// TwinCAT 3 PLC project StudentStation
// ProgramVersion: 3.1.4022.4
// libraries:
//   Tc2_Standard, * (Beckhoff Automation GmbH)
//   Tc2_System, * (Beckhoff Automation GmbH)
//   Tc3_Module, * (Beckhoff Automation GmbH)
//   VisuDialogs, * (System)
//   VisuSymbols,3.5.10.0,System
// project tree:
//   ABBControl/ ABBAssemble.TcPOU (not stored), ABBGotoAGVPos.TcPOU (not stored), ABBGotoBuffer.TcPOU (not stored), ABBGotoHome.TcPOU (not stored), ABBGotoScanner.TcPOU (not stored), ABBGotoTable.TcPOU (not stored), ABBPickLeaveBuffer.TcPOU (not stored), ABBPickLeaveContainerAGV.TcPOU (not stored), ABBPickLeaveContaineronTable.TcPOU (not stored), ABBPickLeaveScanner.TcPOU (not stored), ABBScanContainer.TcPOU (not stored), ABBScannerStation.TcPOU (not stored)
//   Automation Library/ AGVControlSystem.TcPOU (not stored), AutomationLibrary.TcPOU (not stored), BookingSystem.TcPOU (not stored), CommData.TcGVL (not stored), OrderHandling.TcPOU (not stored), PhysicalSystemTest.TcPOU (not stored), RobotControlSystem.TcPOU (not stored), RobotPosTracker.TcPOU (not stored), SensorReader.TcPOU (not stored), Visualaisation_Control.TcPOU (not stored)
//   DUTs/ ABBPositions.TcDUT (not stored), ABBXYPOS.TcDUT (not stored), OrderPLC.TcDUT (not stored), PLCRobotOrder.TcDUT (not stored), Station.TcDUT (not stored), Storage.TcDUT (not stored)
//   / GlobalTextList.TcGTLO, PlcTask.TcTTO (not stored), Visualization Manager.TcVMO (not stored)
//   GVLs/ GVL.TcGVL
//   POUs/ ModeControl.TcPOU, ManualMode.TcPOU, AssembleParts.TcPOU, LoadFromAGV.TcPOU, ScanBuffer.TcPOU, Robot.TcPOU, AutoMode.TcPOU, MAIN.TcPOU, IdentifyPart.TcPOU
//   VISUs/ RobotStation.TcVIS (not stored), Station.TcVIS, Visualization.TcVIS
// real-time tasks:
//   TASK PlcTask: cycle T#10ms, priority 20, ADS port 350

// ---- GVLs/GVL.TcGVL
{attribute 'qualified_only'}
VAR_GLOBAL
	// Order for the next assembly part. The part name should be sent as per the part list and case sensitive. 
	{attribute 'OPC.UA.DA' := '1'}
	qsOrderFornextAssembly AT %Q*: STRING := '0';
	// Parts in your Station buffer. Each buffer have 3 storage locations. The part name and quantity should be mentioned.
	{attribute 'OPC.UA.DA' := '1'}
	BufferProducts AT %Q*: Station;
	// Signal to AGV, a pallet is placed from Station to the AGV. 
	{attribute 'OPC.UA.DA' := '1'}
	qxPalletPlacedinAGV AT %Q*: BOOL;
	// Signal From AGV, that it have docked in your station
	{attribute 'OPC.UA.DA' := '1'}
	ixAGVatStation AT %I*: BOOL;
	// Signal Denoting An AGV have arrived in the Station
	{attribute 'OPC.UA.DA' := '1'}	
	qxPickedfromAGV AT %Q*:BOOL; //Part is picked up from the AGV
	{attribute 'OPC.UA.DA' := '1'}
	mwStationStatus AT %Q*: INT; //Pre-Conditioning Mode //100:Ready to Work § 200: Getting Booked § 300: Booked and Busy § 400 : Manual mode  § 500: Pause Mode § 1000 : Emergency Mode 
	{attribute 'OPC.UA.DA' := '1'}	
	// Emergency Stop is active
	ixEmergencyStop AT %Q*:BOOL;
	
	// Inductive sensor reading. from scaning station
	ixInductiveSensor1 AT %I*:BOOL;
	// Inductive sensor reading. from scaning station
	ixInductiveSensor2 AT %I*:BOOL;
	// Inductive sensor reading. from scaning station
	ixInductiveSensor3 AT %I*:BOOL;
	// Inductive sensor reading. from scaning station
	ixInductiveSensor4 AT %I*:BOOL;
	// Inductive sensor reading. from the sensor in robot Tool
	ixInductiveSensorinTool AT %I*:BOOL;
	// Station ID of the station you are working with.
	{attribute 'OPC.UA.DA' := '1'}
	mwStationID AT %Q*: INT;
	
	sABBFunction : ARRAY [1..12] OF STRING := ['ABBAssemble','ABBGotoAGVPos','ABBGotoBuffer','ABBGotoHome','ABBGotoScanner','ABBGotoTable','ABBPickLeaveBuffer','ABBPickLeaveContainerAGV','ABBPickLeaveContainerOnTable','ABBPickLeaveScanner','ABBScanContainer', 'ABBScannerStation'];
	sBufferIDlist : ARRAY [1..3] OF STRING := ['Storage Position 1','Storage Position 2','Storage Position 3'];
	sPart : ARRAY [1..3] OF STRING := ['Plate','Cylinder','Octagon'];
	sPickOrLeave : ARRAY [1..2] OF STRING := ['Pick','Leave'];
	sABBFunctionList : ARRAY [1..12] OF STRING := ['ABBAssemble','ABBGotoAGVPos','ABBGotoBuffer','ABBGotoHome','ABBGotoScanner','ABBGotoTable','ABBPickLeaveBuffer','ABBPickLeaveContainerAGV','ABBPickLeaveContainerOnTable','ABBPickLeaveScanner','ABBScanContainer', 'ABBScannerStation'];
END_VAR

// ---- POUs/Robot.TcPOU
PROGRAM Robot
VAR
	// Goto Home
	ABBGotoHome_Control: ABBGotoHome;
	GotoHome: BOOL;
	GotoHomeDone: BOOL;
	
	// Go to AGV
	ABBGotoAGVPosByScanner_Control: ABBGotoAGVPos;
	GotoAGVByScanner: BOOL;
	GotoAGVByScannerDone: BOOL;
	
	// Go to AGV
	ABBGotoAGVPosByAssembly_Control: ABBGotoAGVPos;
	GotoAGVByAssembly: BOOL;
	GotoAGVByAssemblyDone: BOOL;
	
	// Go to Scanner
	ABBGotoScannerFromAGV_Control: ABBGotoScanner;
	ABBGotoScannerFromBuffer_Control: ABBGotoScanner;
	GotoScannerFromBuffer: BOOL;
	GotoScannerFromAGV: BOOL;
	GotoScannerFromBufferDone: BOOL;
	GotoScannerFromAGVDone: BOOL;
	
	// Go to Table
	ABBGotoTableByAGV_Control: ABBGotoTable;
	GotoTableByAGV: BOOL;
	GotoTableByAGVDone: BOOL;
	
	ABBGotoTableByScanner_Control: ABBGotoTable;
	GotoTableByScanner: BOOL;
	GotoTableDoneByScanner: BOOL;
	
	ABBGotoTableByAssembly_Control: ABBGotoTable;
	GotoTableByAssembly: BOOL;
	GotoTableDoneByAssembly: BOOL;
	
	// Go to Buffer
	ABBGotoBuffer_Control: ABBGotoBuffer;
	GotoBuffer: BOOL;
	GotoBufferDone: BOOL;
	
	// PickLeave Container AGV
	ABBPickLeaveContainerAGV_Control: ABBPickLeaveContainerAGV;
	PickAGV: BOOL;
	LeaveAGV: BOOL;
	PickLeaveAGVDone: BOOL;
	
	// PickLeave Scanner
	ABBPickLeaveScannerFromBuffer_Control: ABBPickLeaveScanner;
	ABBPickLeaveScannerFromAGV_Control: ABBPickLeaveScanner;
	PickScannerFromBuffer: BOOL;
	LeaveScannerFromBuffer: BOOL;
	PickLeaveScannerFromBufferDone: BOOL;
	PickScannerFromAGV: BOOL;
	LeaveScannerFromAGV: BOOL;
	PickLeaveScannerFromAGVDone: BOOL;
	
	
	// PickLeave Buffer
	ABBPickLeaveBuffer_Control: ABBPickLeaveBuffer;
	PickBuffer: BOOL;
	LeaveBuffer: BOOL;
	PickLeaveBufferDone: BOOL;
	
	// PickLeave Table
	ABBPickLeaveTable_Control: ABBPickLeaveContaineronTable;
	PickTable: BOOL;
	LeaveTable: BOOL;
	PickLeaveTableDone: BOOL;
	
	// Scan parts
	ABBScanContainer_Control: ABBScanContainer;
	ScanContainer: BOOL;
	ScanContainerPartAvailable: BOOL;
	ScanContainerDone: BOOL;
	
	// Assemble parts
	ABBAssemble_Control: ABBAssemble;
	Assemble: BOOL;
	AssembleBufferId: INT;
	AssemblePartId: INT;
	AssembleDone: BOOL;
	
	// Read sensor
	ABBScannerStationByBuffer_Control: ABBScannerStation;
	ABBScannerStationByAGV_Control: ABBScannerStation;
	ReadSensorByBuffer: BOOL;
	ReadSensorByAGV: BOOL;
	ReadSensorByBufferDone: BOOL;
	ReadSensorByAGVDone: BOOL;
	
	
	// Read sensor
	IdentifyPartFB: IdentifyPart;
	IdentifyPart_Control: IdentifyPart;
	ScanPartId: INT;
END_VAR

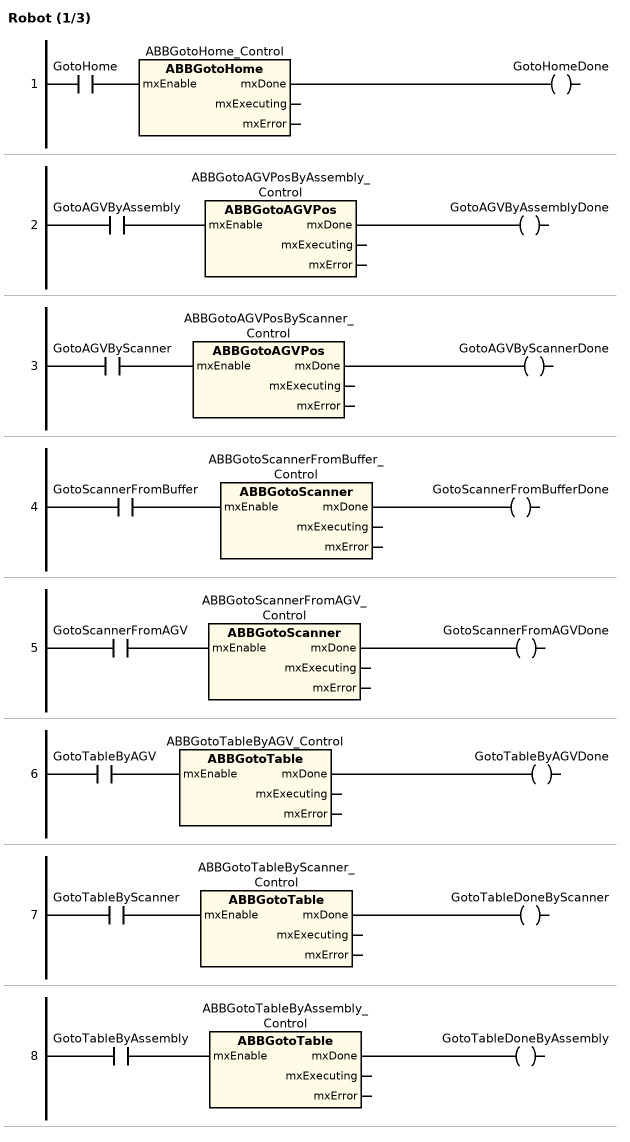
// NETWORK 1
ABBGotoHome_Control(mxEnable := GotoHome); // ABBGotoHome
GotoHomeDone := ABBGotoHome_Control.mxDone;

// NETWORK 2
ABBGotoAGVPosByAssembly_Control(mxEnable := GotoAGVByAssembly); // ABBGotoAGVPos
GotoAGVByAssemblyDone := ABBGotoAGVPosByAssembly_Control.mxDone;

// NETWORK 3
ABBGotoAGVPosByScanner_Control(mxEnable := GotoAGVByScanner); // ABBGotoAGVPos
GotoAGVByScannerDone := ABBGotoAGVPosByScanner_Control.mxDone;

// NETWORK 4
ABBGotoScannerFromBuffer_Control(mxEnable := GotoScannerFromBuffer); // ABBGotoScanner
GotoScannerFromBufferDone := ABBGotoScannerFromBuffer_Control.mxDone;

// NETWORK 5
ABBGotoScannerFromAGV_Control(mxEnable := GotoScannerFromAGV); // ABBGotoScanner
GotoScannerFromAGVDone := ABBGotoScannerFromAGV_Control.mxDone;

// NETWORK 6
ABBGotoTableByAGV_Control(mxEnable := GotoTableByAGV); // ABBGotoTable
GotoTableByAGVDone := ABBGotoTableByAGV_Control.mxDone;

// NETWORK 7
ABBGotoTableByScanner_Control(mxEnable := GotoTableByScanner); // ABBGotoTable
GotoTableDoneByScanner := ABBGotoTableByScanner_Control.mxDone;

// NETWORK 8
ABBGotoTableByAssembly_Control(mxEnable := GotoTableByAssembly); // ABBGotoTable
GotoTableDoneByAssembly := ABBGotoTableByAssembly_Control.mxDone;

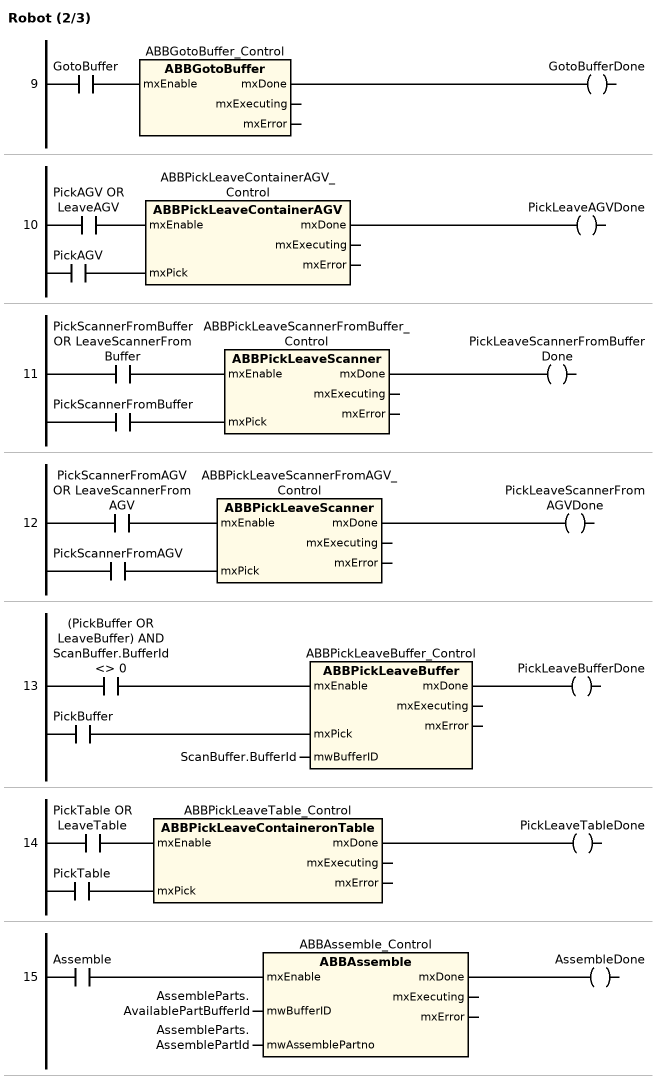
// NETWORK 9
ABBGotoBuffer_Control(mxEnable := GotoBuffer); // ABBGotoBuffer
GotoBufferDone := ABBGotoBuffer_Control.mxDone;

// NETWORK 10
ABBPickLeaveContainerAGV_Control(mxEnable := PickAGV OR LeaveAGV, mxPick := PickAGV); // ABBPickLeaveContainerAGV
PickLeaveAGVDone := ABBPickLeaveContainerAGV_Control.mxDone;

// NETWORK 11
ABBPickLeaveScannerFromBuffer_Control(mxEnable := PickScannerFromBuffer OR LeaveScannerFromBuffer, mxPick := PickScannerFromBuffer); // ABBPickLeaveScanner
PickLeaveScannerFromBufferDone := ABBPickLeaveScannerFromBuffer_Control.mxDone;

// NETWORK 12
ABBPickLeaveScannerFromAGV_Control(mxEnable := PickScannerFromAGV OR LeaveScannerFromAGV, mxPick := PickScannerFromAGV); // ABBPickLeaveScanner
PickLeaveScannerFromAGVDone := ABBPickLeaveScannerFromAGV_Control.mxDone;

// NETWORK 13
ABBPickLeaveBuffer_Control(
    mxEnable := (PickBuffer OR LeaveBuffer) AND ScanBuffer.BufferId <> 0,
    mxPick := PickBuffer,
    mwBufferID := ScanBuffer.BufferId); // ABBPickLeaveBuffer
PickLeaveBufferDone := ABBPickLeaveBuffer_Control.mxDone;

// NETWORK 14
ABBPickLeaveTable_Control(mxEnable := PickTable OR LeaveTable, mxPick := PickTable); // ABBPickLeaveContaineronTable
PickLeaveTableDone := ABBPickLeaveTable_Control.mxDone;

// NETWORK 15
ABBAssemble_Control(
    mxEnable := Assemble,
    mwBufferID := AssembleParts.AvailablePartBufferId,
    mwAssemblePartno := AssembleParts.AssemblePartId); // ABBAssemble
AssembleDone := ABBAssemble_Control.mxDone;

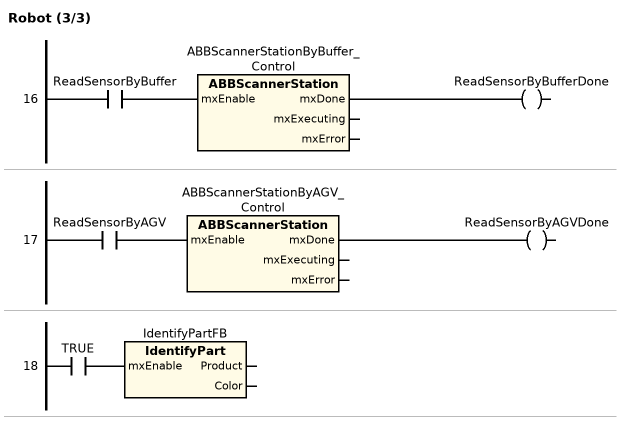
// NETWORK 16
ABBScannerStationByBuffer_Control(mxEnable := ReadSensorByBuffer); // ABBScannerStation
ReadSensorByBufferDone := ABBScannerStationByBuffer_Control.mxDone;

// NETWORK 17
ABBScannerStationByAGV_Control(mxEnable := ReadSensorByAGV); // ABBScannerStation
ReadSensorByAGVDone := ABBScannerStationByAGV_Control.mxDone;

// NETWORK 18
IdentifyPartFB(mxEnable := TRUE); // IdentifyPart

END_PROGRAM

// ---- POUs/IdentifyPart.TcPOU
FUNCTION_BLOCK IdentifyPart
VAR_INPUT
	mxEnable: BOOL;
END_VAR
VAR_OUTPUT
	Product:STRING;
	Color: STRING;
	Component: STRING;
END_VAR
VAR
	SensorReader:BYTE;
END_VAR

IF mxEnable THEN
	SensorReader.1:=gvl.ixInductiveSensor1;
	SensorReader.2:=gvl.ixInductiveSensor2;
	SensorReader.3:=gvl.ixInductiveSensor3;
	SensorReader.4:=gvl.ixInductiveSensor4;
END_IF

IF SensorReader = 0 OR SensorReader = 4 OR SensorReader = 2 OR SensorReader = 6 THEN
 	Product:='InvalidPart';
	Color := '';
	Component := 'invalidpart';
END_IF

IF SensorReader=16 THEN
	Product:='CONTAINER';
	Color := 'BLUE';
	Component := 'BLUECONTAINER';
END_IF

IF SensorReader=8 THEN
	Product:='CONTAINER';
	Color := 'YELLOW';
	Component := 'YELLOWCONTAINER';
END_IF

IF SensorReader=24 THEN
	Product:='CONTAINER';
	Color := 'RED';
	Component := 'REDCONTAINER';
END_IF

IF SensorReader=20 THEN
	Product:='CYLINDER';
	Color := 'BLUE';
	Component := 'BLUECYLINDER';
END_IF

IF SensorReader=12 THEN
	Product:='OCTAGON';
	Color := 'BLUE';
	Component := 'BLUEOCTAGON';
END_IF

IF SensorReader=28 THEN
	Product:='PLATE';
	Color := 'BLUE';
	Component := 'BLUEPLATE';
END_IF

IF SensorReader=18 THEN
	Product:='CYLINDER';
	Color := 'YELLOW';
	Component := 'YELLOWCYLINDER';
END_IF

IF SensorReader=10 THEN
	Product:='OCTAGON';
	Color := 'YELLOW';
	Component := 'YELLOWOCTAGON';
END_IF

IF SensorReader=26 THEN
	Product:='PLATE';
	Color := 'YELLOW';
	Component := 'YELLOWPLATE';
END_IF

IF SensorReader=22 THEN
	Product:='CYLINDER';
	Color := 'RED';
	Component := 'REDCYLINDER';
END_IF

IF SensorReader=14 THEN
	Product:='OCTAGON';
	Color := 'RED';
	Component := 'REDOCTAGON';
END_IF

IF SensorReader=30 THEN
	Product:='PLATE';
	Color := 'RED';
	Component := 'REDPLATE';
END_IF

END_FUNCTION_BLOCK

// ---- POUs/ScanBuffer.TcPOU
PROGRAM ScanBuffer
VAR
	// Default
	Done: BOOL;
	
	// Goto Buffer id
	BufferId: INT;
	BufferIdReady: BOOL;
	
	// Invalid Buffer part
	InvalidPart: BOOL;
	Quatity: INT;
END_VAR

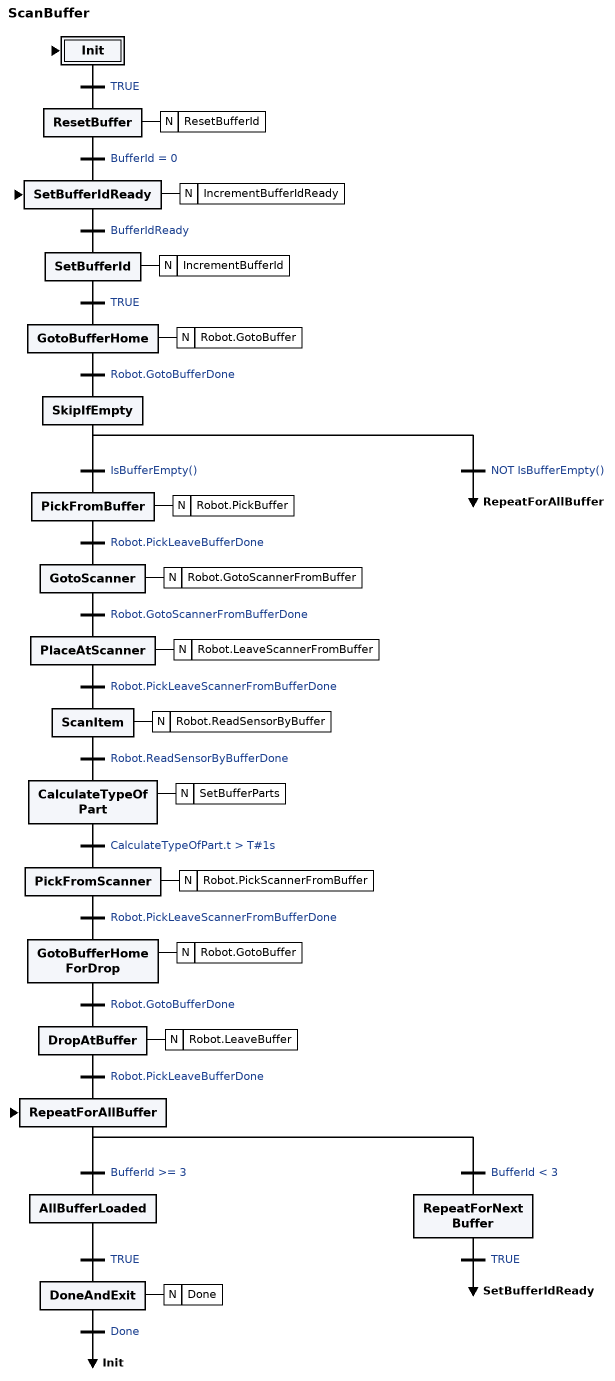
INITIAL_STEP Init:
END_STEP
TRANSITION FROM Init TO ResetBuffer
    := TRUE;
END_TRANSITION
STEP ResetBuffer:
    ResetBufferId(N);
END_STEP
TRANSITION FROM ResetBuffer TO SetBufferIdReady
    := BufferId = 0;
END_TRANSITION
STEP SetBufferIdReady:
    IncrementBufferIdReady(N);
END_STEP
TRANSITION FROM SetBufferIdReady TO SetBufferId
    := BufferIdReady;
END_TRANSITION
STEP SetBufferId:
    IncrementBufferId(N);
END_STEP
TRANSITION FROM SetBufferId TO GotoBufferHome
    := TRUE;
END_TRANSITION
STEP GotoBufferHome:
    Robot.GotoBuffer(N);
END_STEP
TRANSITION FROM GotoBufferHome TO SkipIfEmpty
    := Robot.GotoBufferDone;
END_TRANSITION
STEP SkipIfEmpty:
END_STEP
TRANSITION FROM SkipIfEmpty TO PickFromBuffer
    := IsBufferEmpty();
END_TRANSITION
TRANSITION FROM SkipIfEmpty TO RepeatForAllBuffer
    := NOT IsBufferEmpty();
END_TRANSITION
STEP PickFromBuffer:
    Robot.PickBuffer(N);
END_STEP
TRANSITION FROM PickFromBuffer TO GotoScanner
    := Robot.PickLeaveBufferDone;
END_TRANSITION
STEP GotoScanner:
    Robot.GotoScannerFromBuffer(N);
END_STEP
TRANSITION FROM GotoScanner TO PlaceAtScanner
    := Robot.GotoScannerFromBufferDone;
END_TRANSITION
STEP PlaceAtScanner:
    Robot.LeaveScannerFromBuffer(N);
END_STEP
TRANSITION FROM PlaceAtScanner TO ScanItem
    := Robot.PickLeaveScannerFromBufferDone;
END_TRANSITION
STEP ScanItem:
    Robot.ReadSensorByBuffer(N);
END_STEP
TRANSITION FROM ScanItem TO CalculateTypeOfPart
    := Robot.ReadSensorByBufferDone;
END_TRANSITION
STEP CalculateTypeOfPart:
    SetBufferParts(N);
END_STEP
TRANSITION FROM CalculateTypeOfPart TO PickFromScanner
    := CalculateTypeOfPart.t > T#1s;
END_TRANSITION
STEP PickFromScanner:
    Robot.PickScannerFromBuffer(N);
END_STEP
TRANSITION FROM PickFromScanner TO GotoBufferHomeForDrop
    := Robot.PickLeaveScannerFromBufferDone;
END_TRANSITION
STEP GotoBufferHomeForDrop:
    Robot.GotoBuffer(N);
END_STEP
TRANSITION FROM GotoBufferHomeForDrop TO DropAtBuffer
    := Robot.GotoBufferDone;
END_TRANSITION
STEP DropAtBuffer:
    Robot.LeaveBuffer(N);
END_STEP
TRANSITION FROM DropAtBuffer TO RepeatForAllBuffer
    := Robot.PickLeaveBufferDone;
END_TRANSITION
STEP RepeatForAllBuffer:
END_STEP
TRANSITION FROM RepeatForAllBuffer TO AllBufferLoaded
    := BufferId >= 3;
END_TRANSITION
STEP AllBufferLoaded:
END_STEP
TRANSITION FROM AllBufferLoaded TO DoneAndExit
    := TRUE;
END_TRANSITION
TRANSITION FROM RepeatForAllBuffer TO RepeatForNextBuffer
    := BufferId < 3;
END_TRANSITION
STEP RepeatForNextBuffer:
END_STEP
TRANSITION FROM RepeatForNextBuffer TO SetBufferIdReady
    := TRUE;
END_TRANSITION
STEP DoneAndExit:
    Done(N);
END_STEP
TRANSITION FROM DoneAndExit TO Init
    := Done;
END_TRANSITION

ACTION IncrementBufferId:
IF BufferIdReady = TRUE THEN
	BufferId := BufferId + 1;
	BufferIdReady := FALSE;
END_IF
END_ACTION

ACTION IncrementBufferIdReady:
BufferIdReady := TRUE;
END_ACTION

METHOD IsBufferEmpty : BOOL
VAR_INPUT
END_VAR
CASE BufferId OF
	1:
		IF GVL.BufferProducts.Storage1.Quatity > 0 THEN
			IsBufferEmpty := FALSE;
		ELSE
			IsBufferEmpty := TRUE;
		END_IF
	2:
		IF GVL.BufferProducts.Storage2.Quatity > 0 THEN
			IsBufferEmpty := FALSE;
		ELSE
			IsBufferEmpty := TRUE;
		END_IF
	3:
		IF GVL.BufferProducts.Storage3.Quatity > 0 THEN
			IsBufferEmpty := FALSE;
		ELSE
			IsBufferEmpty := TRUE;
		END_IF
END_CASE
END_METHOD

ACTION ResetBufferId:
BufferId := 0;
END_ACTION

ACTION SetBufferParts:
IF Robot.IdentifyPartFB.Product = 'PLATE' THEN
	Quatity := 2;
ELSIF Robot.IdentifyPartFB.Product = 'CYLINDER' THEN
	Quatity := 4;
ELSIF Robot.IdentifyPartFB.Product = 'OCTAGON' THEN
	Quatity := 4;
ELSE
	Quatity := 0;
	GVL.mwStationStatus := 1000;
	
END_IF

CASE BufferId OF
	1:
		GVL.BufferProducts.Storage1.Quatity := Quatity;
		GVL.BufferProducts.Storage1.Component := Robot.IdentifyPartFB.Component;
	2:
		GVL.BufferProducts.Storage2.Quatity := Quatity;
		GVL.BufferProducts.Storage2.Component := Robot.IdentifyPartFB.Component;
	3:
		GVL.BufferProducts.Storage3.Quatity := Quatity;
		GVL.BufferProducts.Storage3.Component := Robot.IdentifyPartFB.Component;
END_CASE
END_ACTION

ACTION SkipScan:
GVL.BufferProducts.Storage1.Component := 'REDPLATE';
GVL.BufferProducts.Storage1.Quatity := 2;
GVL.BufferProducts.Storage2.Component := 'REDCYLINDER';
GVL.BufferProducts.Storage2.Quatity := 4;
GVL.BufferProducts.Storage3.Component := 'REDOCTAGON';
GVL.BufferProducts.Storage3.Quatity := 4;
END_ACTION

END_PROGRAM

// ---- POUs/AssembleParts.TcPOU
PROGRAM AssembleParts
VAR
	// Default
	Done: BOOL;
	
	// Scan part id
	AssemblePartId: INT;
	AssemblePartIdReady: BOOL;
	AvailablePartBufferId: INT;
	
	AssembledParts: ARRAY[1..3] OF BOOL;
	
	PartNeedToAssemble: STRING;
	InvalidPart: BOOL;
	Quatity: INT;
	IsUpdateAssemblePartsReady: BOOL;
END_VAR

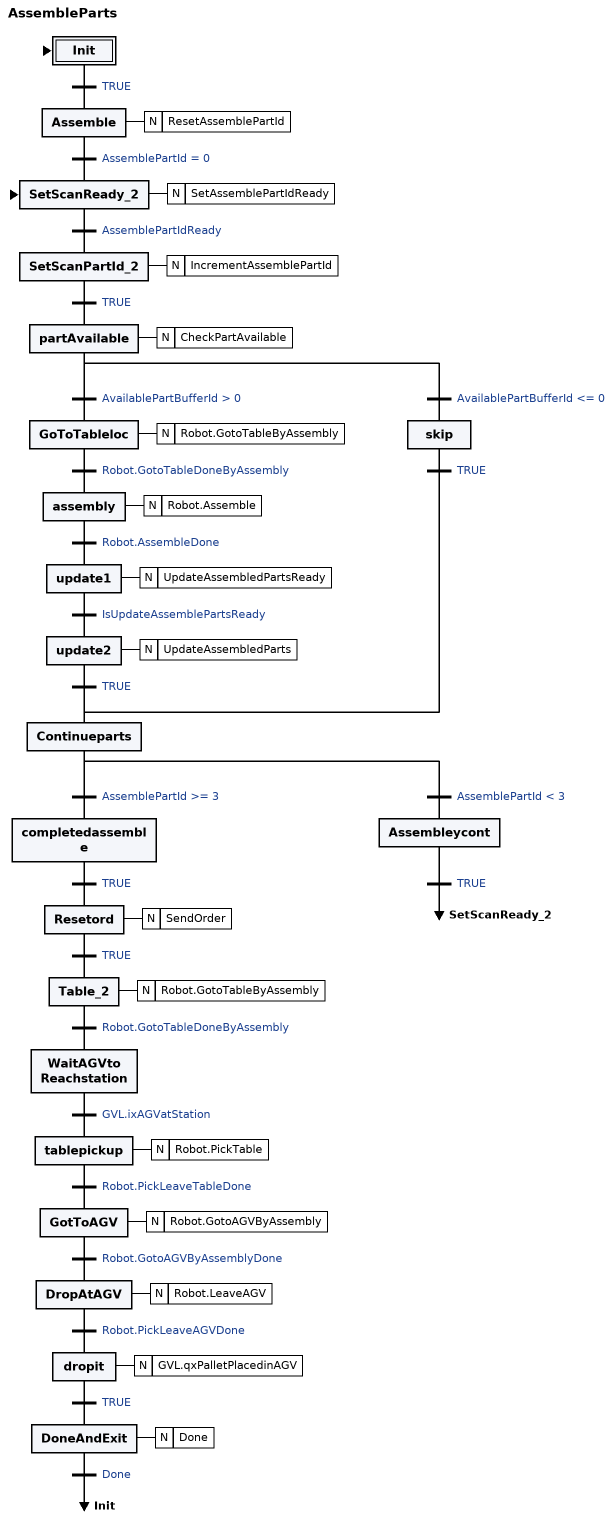
INITIAL_STEP Init:
END_STEP
TRANSITION FROM Init TO Assemble
    := TRUE;
END_TRANSITION
STEP Assemble:
    ResetAssemblePartId(N);
END_STEP
TRANSITION FROM Assemble TO SetScanReady_2
    := AssemblePartId = 0;
END_TRANSITION
STEP SetScanReady_2:
    SetAssemblePartIdReady(N);
END_STEP
TRANSITION FROM SetScanReady_2 TO SetScanPartId_2
    := AssemblePartIdReady;
END_TRANSITION
STEP SetScanPartId_2:
    IncrementAssemblePartId(N);
END_STEP
TRANSITION FROM SetScanPartId_2 TO partAvailable
    := TRUE;
END_TRANSITION
STEP partAvailable:
    CheckPartAvailable(N);
END_STEP
TRANSITION FROM partAvailable TO GoToTableloc
    := AvailablePartBufferId > 0;
END_TRANSITION
STEP GoToTableloc:
    Robot.GotoTableByAssembly(N);
END_STEP
TRANSITION FROM GoToTableloc TO assembly
    := Robot.GotoTableDoneByAssembly;
END_TRANSITION
STEP assembly:
    Robot.Assemble(N);
END_STEP
TRANSITION FROM assembly TO update1
    := Robot.AssembleDone;
END_TRANSITION
STEP update1:
    UpdateAssembledPartsReady(N);
END_STEP
TRANSITION FROM update1 TO update2
    := IsUpdateAssemblePartsReady;
END_TRANSITION
STEP update2:
    UpdateAssembledParts(N);
END_STEP
TRANSITION FROM update2 TO Continueparts
    := TRUE;
END_TRANSITION
TRANSITION FROM partAvailable TO skip
    := AvailablePartBufferId <= 0;
END_TRANSITION
STEP skip:
END_STEP
TRANSITION FROM skip TO Continueparts
    := TRUE;
END_TRANSITION
STEP Continueparts:
END_STEP
TRANSITION FROM Continueparts TO completedassemble
    := AssemblePartId >= 3;
END_TRANSITION
STEP completedassemble:
END_STEP
TRANSITION FROM completedassemble TO Resetord
    := TRUE;
END_TRANSITION
STEP Resetord:
    SendOrder(N);
END_STEP
TRANSITION FROM Resetord TO Table_2
    := TRUE;
END_TRANSITION
STEP Table_2:
    Robot.GotoTableByAssembly(N);
END_STEP
TRANSITION FROM Table_2 TO WaitAGVtoReachstation
    := Robot.GotoTableDoneByAssembly;
END_TRANSITION
STEP WaitAGVtoReachstation:
END_STEP
TRANSITION FROM WaitAGVtoReachstation TO tablepickup
    := GVL.ixAGVatStation;
END_TRANSITION
STEP tablepickup:
    Robot.PickTable(N);
END_STEP
TRANSITION FROM tablepickup TO GotToAGV
    := Robot.PickLeaveTableDone;
END_TRANSITION
STEP GotToAGV:
    Robot.GotoAGVByAssembly(N);
END_STEP
TRANSITION FROM GotToAGV TO DropAtAGV
    := Robot.GotoAGVByAssemblyDone;
END_TRANSITION
STEP DropAtAGV:
    Robot.LeaveAGV(N);
END_STEP
TRANSITION FROM DropAtAGV TO dropit
    := Robot.PickLeaveAGVDone;
END_TRANSITION
STEP dropit:
    GVL.qxPalletPlacedinAGV(N);
END_STEP
TRANSITION FROM dropit TO DoneAndExit
    := TRUE;
END_TRANSITION
TRANSITION FROM Continueparts TO Assembleycont
    := AssemblePartId < 3;
END_TRANSITION
STEP Assembleycont:
END_STEP
TRANSITION FROM Assembleycont TO SetScanReady_2
    := TRUE;
END_TRANSITION
STEP DoneAndExit:
    Done(N);
END_STEP
TRANSITION FROM DoneAndExit TO Init
    := Done;
END_TRANSITION

ACTION CheckPartAvailable:
CASE AssemblePartId OF
	1:
		PartNeedToAssemble := CONCAT (LoadFromAGV.ContainerColor, 'PLATE');
	2:
		IF AssembledParts[1] THEN
			PartNeedToAssemble := CONCAT (LoadFromAGV.ContainerColor, 'CYLINDER');
		ELSE
			PartNeedToAssemble := 'INVALID';
		END_IF
	3:
		IF AssembledParts[1] THEN
			PartNeedToAssemble := CONCAT (LoadFromAGV.ContainerColor, 'OCTAGON');
		ELSE
			PartNeedToAssemble := 'INVALID';
		END_IF
END_CASE
IF GVL.BufferProducts.Storage1.Component = PartNeedToAssemble AND GVL.BufferProducts.Storage1.Quatity > 0 THEN
	AvailablePartBufferId := 1;
ELSIF GVL.BufferProducts.Storage2.Component = PartNeedToAssemble AND GVL.BufferProducts.Storage2.Quatity > 0 THEN
	AvailablePartBufferId := 2;
ELSIF GVL.BufferProducts.Storage3.Component = PartNeedToAssemble AND GVL.BufferProducts.Storage3.Quatity > 0 THEN
	AvailablePartBufferId := 3;
ELSE
	AvailablePartBufferId := -1;
END_IF
END_ACTION

ACTION IncrementAssemblePartId:
IF AssemblePartIdReady THEN
	AssemblePartId := AssemblePartId + 1;
	AssemblePartIdReady := FALSE;
END_IF
END_ACTION

ACTION ResetAssemblePartId:
AssemblePartId := 0;
AssembledParts[1] := FALSE;
AssembledParts[2] := FALSE;
AssembledParts[3] := FALSE;
END_ACTION

ACTION SendOrder:
IF NOT AssembledParts[1] THEN
	GVL.qsOrderFornextAssembly := CONCAT (LoadFromAGV.ContainerColor, 'PLATE');
ELSIF NOT AssembledParts[2] THEN
	GVL.qsOrderFornextAssembly := CONCAT (LoadFromAGV.ContainerColor, 'CYLINDER');
ELSIF NOT AssembledParts[3] THEN
	GVL.qsOrderFornextAssembly := CONCAT (LoadFromAGV.ContainerColor, 'OCTAGON');
ELSE
	GVL.qsOrderFornextAssembly := 'AssembledProduct';
END_IF
END_ACTION

ACTION SetAssemblePartIdReady:
AssemblePartIdReady := TRUE;
END_ACTION

ACTION UpdateAssembledParts:
IF IsUpdateAssemblePartsReady THEN
	CASE AssemblePartId OF
		1:
			AssembledParts[1] := TRUE;
		2:
			AssembledParts[2] := TRUE;
		3:
			AssembledParts[3] := TRUE;
	END_CASE
	CASE AvailablePartBufferId OF
		1:
			GVL.BufferProducts.Storage1.Quatity := GVL.BufferProducts.Storage1.Quatity - 1;
		2:
			GVL.BufferProducts.Storage2.Quatity := GVL.BufferProducts.Storage2.Quatity - 1;
		3:
			GVL.BufferProducts.Storage3.Quatity := GVL.BufferProducts.Storage3.Quatity - 1;
	END_CASE
	IsUpdateAssemblePartsReady := FALSE;
END_IF
END_ACTION

ACTION UpdateAssembledPartsReady:
IsUpdateAssemblePartsReady := TRUE;
END_ACTION

END_PROGRAM

// ---- POUs/LoadFromAGV.TcPOU
PROGRAM LoadFromAGV
VAR
	// Default
	Done: BOOL;
	
	// Container
	InvalidAGVPart: BOOL;
	ContainerColor: STRING;
	Debug: BOOL;
END_VAR

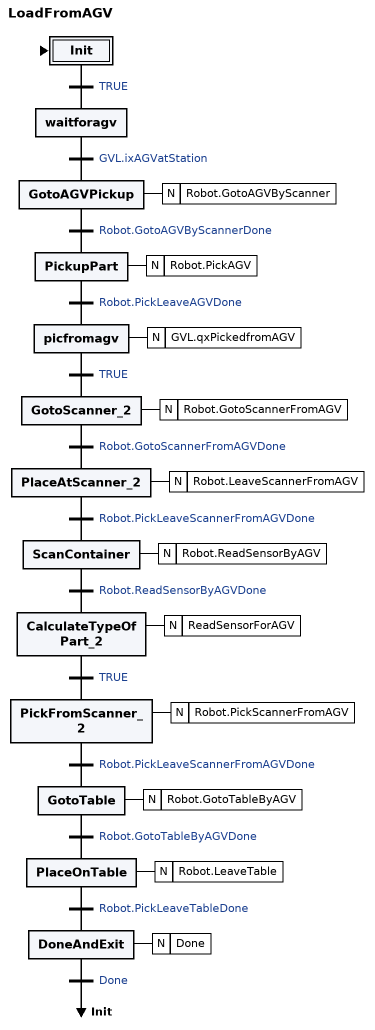
INITIAL_STEP Init:
END_STEP
TRANSITION FROM Init TO waitforagv
    := TRUE;
END_TRANSITION
STEP waitforagv:
END_STEP
TRANSITION FROM waitforagv TO GotoAGVPickup
    := GVL.ixAGVatStation;
END_TRANSITION
STEP GotoAGVPickup:
    Robot.GotoAGVByScanner(N);
END_STEP
TRANSITION FROM GotoAGVPickup TO PickupPart
    := Robot.GotoAGVByScannerDone;
END_TRANSITION
STEP PickupPart:
    Robot.PickAGV(N);
END_STEP
TRANSITION FROM PickupPart TO picfromagv
    := Robot.PickLeaveAGVDone;
END_TRANSITION
STEP picfromagv:
    GVL.qxPickedfromAGV(N);
END_STEP
TRANSITION FROM picfromagv TO GotoScanner_2
    := TRUE;
END_TRANSITION
STEP GotoScanner_2:
    Robot.GotoScannerFromAGV(N);
END_STEP
TRANSITION FROM GotoScanner_2 TO PlaceAtScanner_2
    := Robot.GotoScannerFromAGVDone;
END_TRANSITION
STEP PlaceAtScanner_2:
    Robot.LeaveScannerFromAGV(N);
END_STEP
TRANSITION FROM PlaceAtScanner_2 TO ScanContainer
    := Robot.PickLeaveScannerFromAGVDone;
END_TRANSITION
STEP ScanContainer:
    Robot.ReadSensorByAGV(N);
END_STEP
TRANSITION FROM ScanContainer TO CalculateTypeOfPart_2
    := Robot.ReadSensorByAGVDone;
END_TRANSITION
STEP CalculateTypeOfPart_2:
    ReadSensorForAGV(N);
END_STEP
TRANSITION FROM CalculateTypeOfPart_2 TO PickFromScanner_2
    := TRUE;
END_TRANSITION
STEP PickFromScanner_2:
    Robot.PickScannerFromAGV(N);
END_STEP
TRANSITION FROM PickFromScanner_2 TO GotoTable
    := Robot.PickLeaveScannerFromAGVDone;
END_TRANSITION
STEP GotoTable:
    Robot.GotoTableByAGV(N);
END_STEP
TRANSITION FROM GotoTable TO PlaceOnTable
    := Robot.GotoTableByAGVDone;
END_TRANSITION
STEP PlaceOnTable:
    Robot.LeaveTable(N);
END_STEP
TRANSITION FROM PlaceOnTable TO DoneAndExit
    := Robot.PickLeaveTableDone;
END_TRANSITION
STEP DoneAndExit:
    Done(N);
END_STEP
TRANSITION FROM DoneAndExit TO Init
    := Done;
END_TRANSITION

ACTION ReadSensorForAGV:
ContainerColor := Robot.IdentifyPartFB.Color;
IF Robot.IdentifyPartFB.Product <> 'CONTAINER' THEN
	GVL.mwStationStatus := 1000;
	GVL.ixEmergencyStop := TRUE;
END_IF
END_ACTION

ACTION SkipScan:
ContainerColor:= 'RED';
Debug:= TRUE;
END_ACTION

END_PROGRAM

// ---- POUs/ModeControl.TcPOU
PROGRAM ModeControl
VAR
	AutoModeButtonClick: BOOL;
	AutoMode: BOOL;
	ManualModeButtonClick: BOOL;
	ManualMode: BOOL;
END_VAR

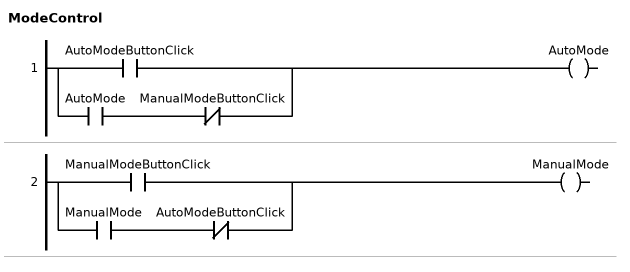
// NETWORK 1
AutoMode := AutoModeButtonClick OR AutoMode AND NOT ManualModeButtonClick;

// NETWORK 2
ManualMode := ManualModeButtonClick OR ManualMode AND NOT AutoModeButtonClick;

END_PROGRAM

// ---- POUs/AutoMode.TcPOU
 PROGRAM AutoMode
VAR
END_VAR

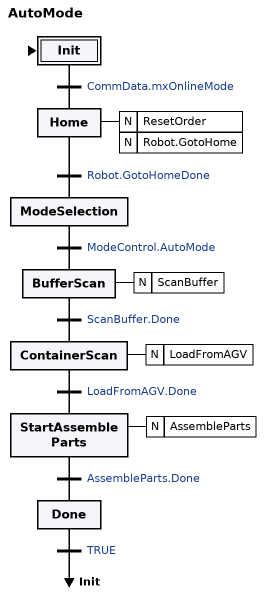
INITIAL_STEP Init:
END_STEP
TRANSITION FROM Init TO Home
    := CommData.mxOnlineMode;
END_TRANSITION
STEP Home:
    ResetOrder(N);
    Robot.GotoHome(N);
END_STEP
TRANSITION FROM Home TO ModeSelection
    := Robot.GotoHomeDone;
END_TRANSITION
STEP ModeSelection:
END_STEP
TRANSITION FROM ModeSelection TO BufferScan
    := ModeControl.AutoMode;
END_TRANSITION
STEP BufferScan:
    ScanBuffer(N);
END_STEP
TRANSITION FROM BufferScan TO ContainerScan
    := ScanBuffer.Done;
END_TRANSITION
STEP ContainerScan:
    LoadFromAGV(N);
END_STEP
TRANSITION FROM ContainerScan TO StartAssembleParts
    := LoadFromAGV.Done;
END_TRANSITION
STEP StartAssembleParts:
    AssembleParts(N);
END_STEP
TRANSITION FROM StartAssembleParts TO Done
    := AssembleParts.Done;
END_TRANSITION
STEP Done:
END_STEP
TRANSITION FROM Done TO Init
    := TRUE;
END_TRANSITION

ACTION ResetOrder:
GVL.qsOrderFornextAssembly := '0';
END_ACTION

ACTION ResetVars:
GVL.BufferProducts.Storage1.Component := '';
GVL.BufferProducts.Storage1.Quatity := 0;
GVL.BufferProducts.Storage2.Component := '';
GVL.BufferProducts.Storage2.Quatity := 0;
GVL.BufferProducts.Storage3.Component := '';
GVL.BufferProducts.Storage3.Quatity := 0;
END_ACTION

END_PROGRAM

// ---- POUs/ManualMode.TcPOU
PROGRAM ManualMode
VAR
	ABBFunction: INT;
	PickLeave: INT;
	BufferID: INT;
	Part: INT;

	Execute: BOOL;
	mxExecute: BOOL;
	
	AssebmleExecuting: BOOL;
	GotoAGVExecuting: BOOL;
	GotoBufferExecuting: BOOL;
	GotoHomeExecuting: BOOL;
	GotoScannerExecuting: BOOL;
	GotoTableExecuting: BOOL;
	PickLeaveBufferExecuting: BOOL;
	PickLeaveContainerExecuting: BOOL;
	PickLeaveContaineronTableExecuting: BOOL;
	PickLeaveScannerExecuting: BOOL;
	ScanContainerExecuting: BOOL;
	ScannerStationExecuting: BOOL;
	
	AssebmleError: BOOL;
	GotoAGVError: BOOL;
	GotoBufferError: BOOL;
	GotoHomeError: BOOL;
	GotoScannerError: BOOL;
	GotoTableError: BOOL;
	PickLeaveBufferError: BOOL;
	PickLeaveContainerError: BOOL;
	PickLeaveContaineronTableError: BOOL;
	PickLeaveScannerError: BOOL;
	ScanContainerError: BOOL;
	ScannerStationError: BOOL;
	
	ABBAssemble_Manual: ABBAssemble;
	ABBGotoAGVPos_Manual: ABBGotoAGVPos;
	ABBGotoBuffer_Manual: ABBGotoBuffer;
	ABBGotoHome_Manual: ABBGotoHome;
	ABBGotoScanner_Manual: ABBGotoScanner;
	ABBGotoTable_Manual: ABBGotoTable;
	ABBPickLeaveBuffer_Manual: ABBPickLeaveBuffer;
	ABBPickLeaveContainerAGV_Manual: ABBPickLeaveContainerAGV;
	ABBPickLeaveContaineronTable_Manual: ABBPickLeaveContaineronTable;
	ABBPickLeaveScanner_Manual: ABBPickLeaveScanner;
	ABBScanContainer_Manual: ABBScanContainer;
	ABBScannerStation_Manual: ABBScannerStation;
END_VAR

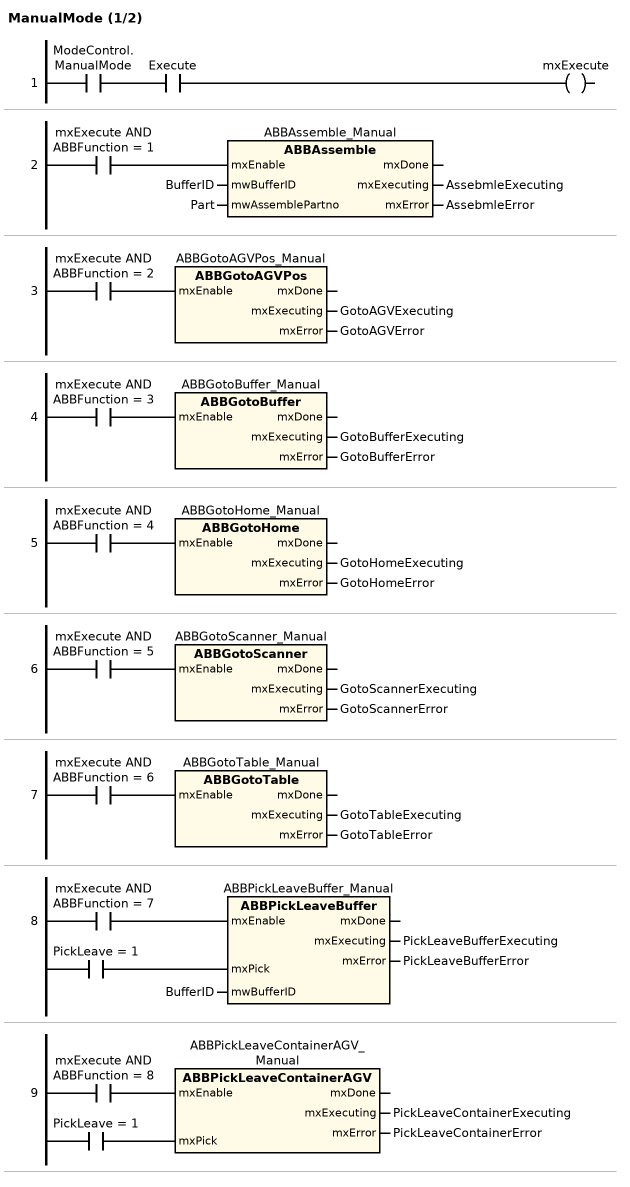
// NETWORK 1
mxExecute := ModeControl.ManualMode AND Execute;

// NETWORK 2
ABBAssemble_Manual(
    mxEnable := mxExecute AND ABBFunction = 1,
    mwBufferID := BufferID,
    mwAssemblePartno := Part,
    mxExecuting => AssebmleExecuting,
    mxError => AssebmleError); // ABBAssemble

// NETWORK 3
ABBGotoAGVPos_Manual(
    mxEnable := mxExecute AND ABBFunction = 2,
    mxExecuting => GotoAGVExecuting,
    mxError => GotoAGVError); // ABBGotoAGVPos

// NETWORK 4
ABBGotoBuffer_Manual(
    mxEnable := mxExecute AND ABBFunction = 3,
    mxExecuting => GotoBufferExecuting,
    mxError => GotoBufferError); // ABBGotoBuffer

// NETWORK 5
ABBGotoHome_Manual(
    mxEnable := mxExecute AND ABBFunction = 4,
    mxExecuting => GotoHomeExecuting,
    mxError => GotoHomeError); // ABBGotoHome

// NETWORK 6
ABBGotoScanner_Manual(
    mxEnable := mxExecute AND ABBFunction = 5,
    mxExecuting => GotoScannerExecuting,
    mxError => GotoScannerError); // ABBGotoScanner

// NETWORK 7
ABBGotoTable_Manual(
    mxEnable := mxExecute AND ABBFunction = 6,
    mxExecuting => GotoTableExecuting,
    mxError => GotoTableError); // ABBGotoTable

// NETWORK 8
ABBPickLeaveBuffer_Manual(
    mxEnable := mxExecute AND ABBFunction = 7,
    mxPick := PickLeave = 1,
    mwBufferID := BufferID,
    mxExecuting => PickLeaveBufferExecuting,
    mxError => PickLeaveBufferError); // ABBPickLeaveBuffer

// NETWORK 9
ABBPickLeaveContainerAGV_Manual(
    mxEnable := mxExecute AND ABBFunction = 8,
    mxPick := PickLeave = 1,
    mxExecuting => PickLeaveContainerExecuting,
    mxError => PickLeaveContainerError); // ABBPickLeaveContainerAGV

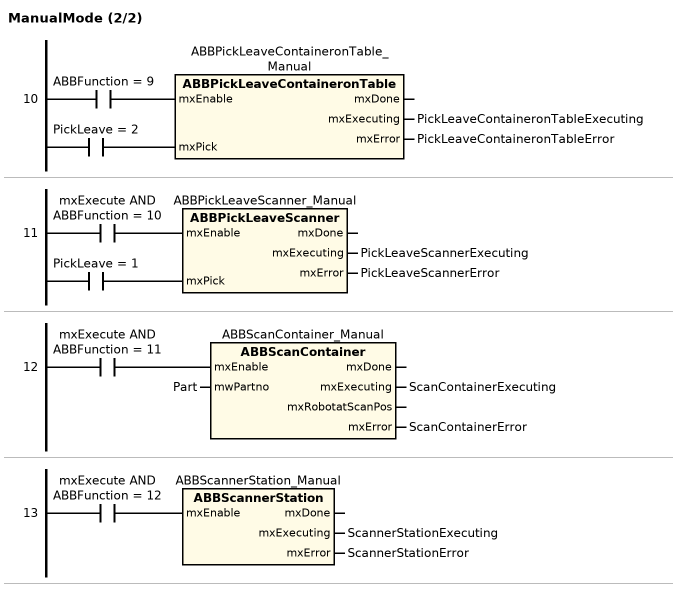
// NETWORK 10
ABBPickLeaveContaineronTable_Manual(
    mxEnable := ABBFunction = 9,
    mxPick := PickLeave = 2,
    mxExecuting => PickLeaveContaineronTableExecuting,
    mxError => PickLeaveContaineronTableError); // ABBPickLeaveContaineronTable

// NETWORK 11
ABBPickLeaveScanner_Manual(
    mxEnable := mxExecute AND ABBFunction = 10,
    mxPick := PickLeave = 1,
    mxExecuting => PickLeaveScannerExecuting,
    mxError => PickLeaveScannerError); // ABBPickLeaveScanner

// NETWORK 12
ABBScanContainer_Manual(
    mxEnable := mxExecute AND ABBFunction = 11,
    mwPartno := Part,
    mxExecuting => ScanContainerExecuting,
    mxError => ScanContainerError); // ABBScanContainer

// NETWORK 13
ABBScannerStation_Manual(
    mxEnable := mxExecute AND ABBFunction = 12,
    mxExecuting => ScannerStationExecuting,
    mxError => ScannerStationError); // ABBScannerStation

END_PROGRAM

// ---- POUs/MAIN.TcPOU
PROGRAM MAIN
VAR
END_VAR

AutomationLibrary();
Visualaisation_Control();
RobotPosTracker();

Robot();
AutoMode();
ModeControl();
ManualMode();

END_PROGRAM

// ---- GlobalTextList.TcGTLO
TEXTLIST GlobalTextList
  153 = ' %s'
  135 = '%s'
  875 = '1'
  207 = '2'
  492 = '21'
  288 = '3'
  431 = 'ABB '
  988 = 'ABB Functions'
  435 = 'AGV'
  139 = 'AGV at Station :'
  375 = 'AGV Scan Table'
  171 = 'All Buffer Check'
  575 = 'All Home Check'
  974 = 'Aseembly'
  126 = 'Assemble'
  578 = 'Assembly Status'
  407 = 'Auto'
  941 = 'AUTO'
  761 = 'AUTO MODE'
  641 = 'Booking from IO Station  :'
  16 = 'Buffer'
  744 = 'BUFFER'
  85 = 'Buffer 1'
  300 = 'Buffer 2'
  301 = 'Buffer 3'
  684 = 'Buffer ID'
  25 = 'BufferID'
  621 = 'Color'
  728 = 'Container'
  932 = 'CONTAINER'
  448 = 'Container Color'
  281 = 'Control for Station'
  704 = 'Cyclinder'
  479 = 'CYLINDER'
  150 = 'Debug Mode'
  228 = 'DebugMode'
  379 = 'Dummy BUffer'
  698 = 'Dummy Buffer'
  390 = 'Emergency Mode'
  137 = 'Emergency Signal :'
  493 = 'Emergency Stop'
  136 = 'Error from Comm :'
  283 = 'Execute'
  250 = 'EXECUTE'
  170 = 'Gabriel Sebastian'
  751 = 'Gabriel Sebastian gabriel.sebastian@hv.se'
  995 = 'Gabriel Sebastian | gabriel.sebastian@hv.se'
  701 = 'Gabriel Sebastian |gabriel.sebastian@hv.se'
  688 = 'Gripper Control'
  247 = 'Gripper Toggle'
  140 = 'Inventory Status'
  395 = 'ixAGVatStation'
  803 = 'Label'
  498 = 'Leave at AGV'
  298 = 'Main Menu'
  731 = 'Manual'
  626 = 'MANUAL'
  917 = 'Manual Controller'
  421 = 'MANUAL MODE'
  203 = 'New AGV to Station :'
  151 = 'Normal Mode'
  478 = 'Octagon'
  770 = 'OCTAGON'
  287 = 'OFF'
  363 = 'Offline'
  741 = 'OFFLINE'
  374 = 'ON'
  13 = 'Online'
  979 = 'ONLINE'
  174 = 'Order for Next Assembly  : %s'
  138 = 'Pallet Placed on AGV :'
  147 = 'Pallet Sensor 1  :'
  146 = 'Pallet Sensor 2  :'
  148 = 'Pallet Sensor 3  :'
  145 = 'Pallet Sensor 4  :'
  114 = 'Part'
  130 = 'PART IDENTIFY'
  213 = 'PartID'
  900 = 'PARTIDENTIFY'
  530 = 'PICK OR LEAVE'
  278 = 'Pick/Leave'
  113 = 'Plate'
  401 = 'PLATE'
  669 = 'PLC'
  733 = 'Quanitity'
  196 = 'Request Generator'
  556 = 'Robot'
  625 = 'Robot Position  : %s'
  881 = 'Robot Power'
  502 = 'Robot Station'
  620 = 'Scan Container'
  204 = 'Scanner'
  899 = 'Sensor Reading  : %s'
  238 = 'Sensor Reading completed'
  144 = 'Sensor Signals'
  134 = 'Station ID :'
  152 = 'Station Offline'
  494 = 'Station Status  : %s'
  458 = 'Station View'
  895 = 'STATUS'
  143 = 'Storage Pos 1: %s'
  141 = 'Storage Pos 2: %s'
  142 = 'Storage Pos 3: %s'
  266 = 'Table To AGV'
  309 = 'Test System'
  149 = 'Tool Sensor  :'
  679 = 'TOTALQUANTITY'
  886 = 'Visualization'
  127 = 'X  : %s'
  412 = 'Y  : %s'
END_TEXTLIST

// ---- VISUs/Station.TcVIS
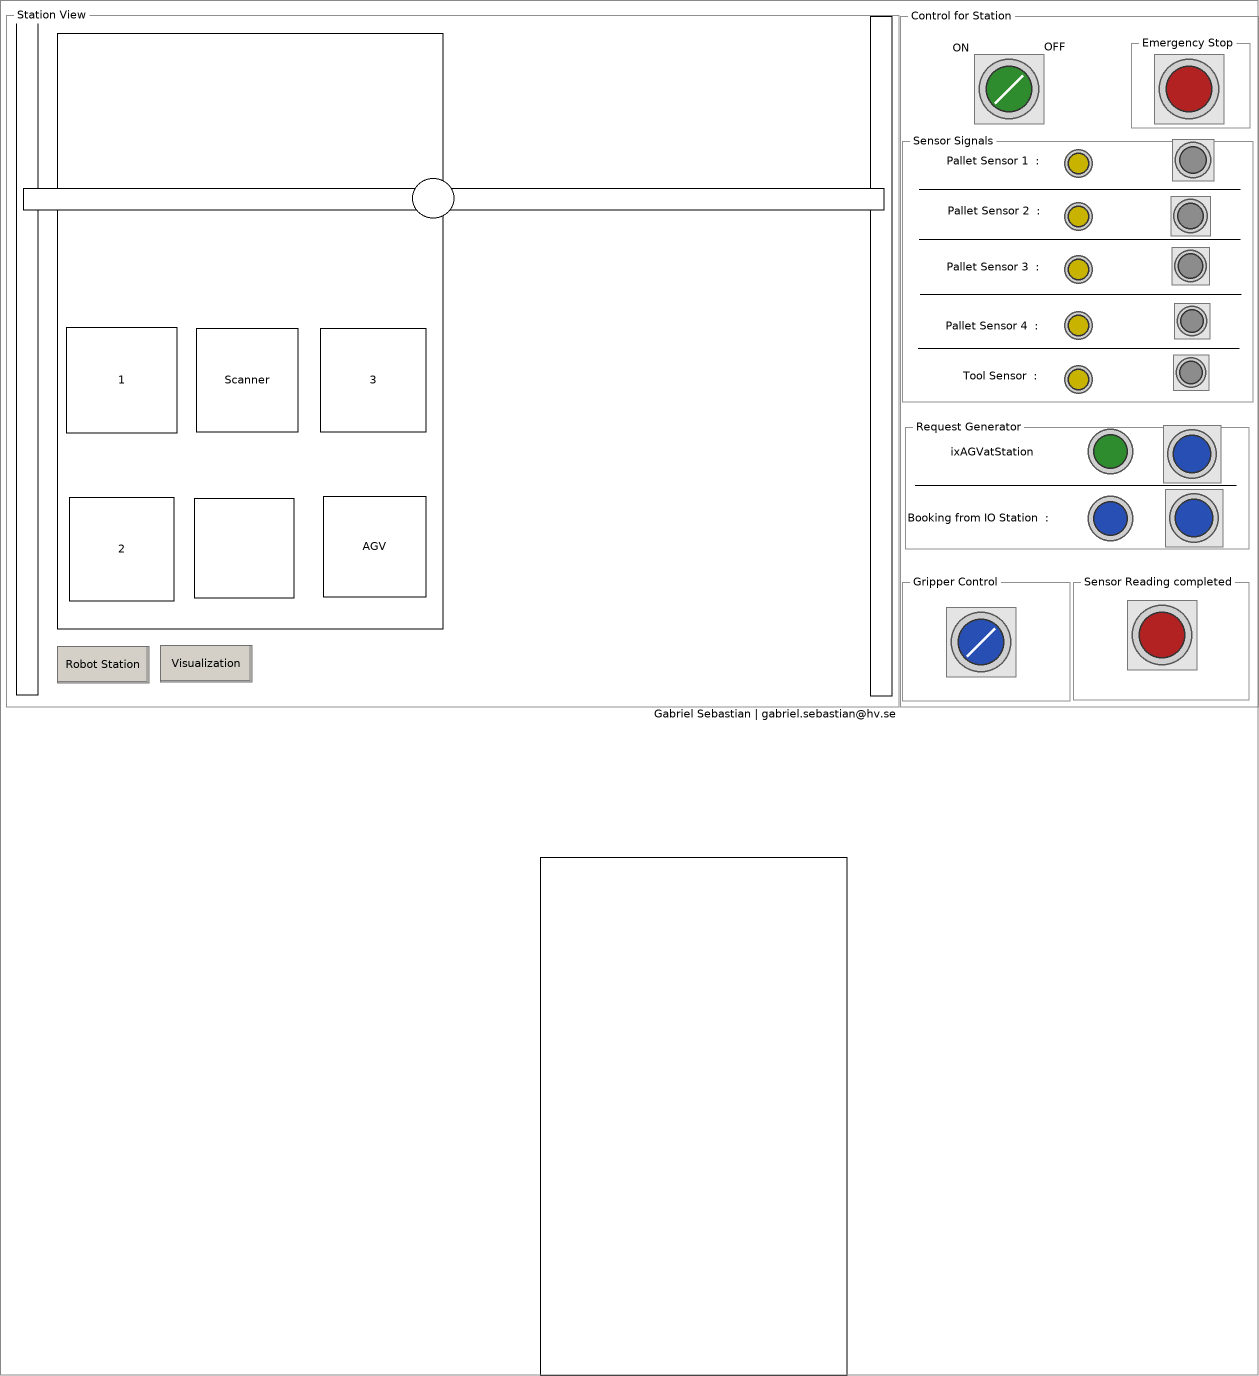
VISUALIZATION Station  // 1259x1376
    RoundedRectangle (540,857 307x519)
        p2738717112: CommData.mwCurrentAGVPOS
    Rectangle (16,15 22x680)
    GroupBox (6,7 893x700), "Station View"
        Rectangle (51,26 386x596)
        Rectangle (864,9 22x680)
        Rectangle (188,491 100x100)
        Rectangle (317,489 103x101), "AGV"
        Rectangle (190,321 102x104), "Scanner"
        Rectangle (60,320 111x106), "1"
        Rectangle (314,321 106x104), "3"
        Rectangle (63,490 105x104), "2"
        RoundedRectangle (17,181 861x22)
            p2738717112: CommData.mwYaxis
        Ellipse (406,171 42x40)
            p2738717112: CommData.mwYaxis
            p3560616238: CommData.mwXaxis
        Button (154,638 92x37), "Visualization"
            OnMouseClick: change screen: Visualization
        Button (51,639 92x37), "Robot Station"
            OnMouseClick: change screen: RobotStation
    GroupBox (900,8 359x699), "Control for Station"
        GroupBox (2,125 351x269), "Sensor Signals"
            Label (15,178 150x30), "Pallet Sensor 4 :"
            Label (17,63 150x30), "Pallet Sensor 2 :"
            Label (16,13 150x30), "Pallet Sensor 1 :"
            Line (17,56) (338,56)
            Lamp1 (160,14 33x33), variable: GVL.ixInductiveSensor1, style: Lamp-Lamp1-Yellow
            Lamp1 (160,67 33x33), variable: GVL.ixInductiveSensor2, style: Lamp-Lamp1-Yellow
            Lamp1 (160,120 33x33), variable: GVL.ixInductiveSensor3, style: Lamp-Lamp1-Yellow
            Lamp1 (160,176 33x33), variable: GVL.ixInductiveSensor4, style: Lamp-Lamp1-Yellow
            Label (16,119 150x30), "Pallet Sensor 3 :"
            Label (23,228 150x30), "Tool Sensor :"
            Lamp1 (160,230 33x33), variable: GVL.ixInductiveSensorinTool, style: Lamp-Lamp1-Yellow
            PushSwitch (266,6 50x42), variable: GVL.ixInductiveSensor1, input disabled if: CommData.mxRobotOnline, behaviour: TOGGLE, style: Switch-PushSwitch-Gray
            PushSwitch (267,63 43x40), variable: GVL.ixInductiveSensor2, input disabled if: CommData.mxRobotOnline, behaviour: TOGGLE, style: Switch-PushSwitch-Gray
            PushSwitch (270,170 40x36), variable: GVL.ixInductiveSensor4, input disabled if: CommData.mxRobotOnline, behaviour: TOGGLE, style: Switch-PushSwitch-Gray
            PushSwitch (271,221 36x37), variable: GVL.ixInductiveSensorinTool, input disabled if: CommData.mxRobotOnline, behaviour: TOGGLE, style: Switch-PushSwitch-Gray
            Line (17,106) (338,106)
            Line (18,161) (339,161)
            Line (16,215) (337,215)
            PushSwitch (269,114 39x38), variable: GVL.ixInductiveSensor3, input disabled if: CommData.mxRobotOnline, behaviour: TOGGLE, style: Switch-PushSwitch-Gray
        RotarySwitch (74,46 70x70), variable: CommData.mxOnlineMode, invisible if: CommData.mxRobotOnline, behaviour: TOGGLE, style: Switch-RotarySwitch-Green
        Label (106,24 98x30), "OFF", invisible if: CommData.mxRobotOnline
        Label (12,25 98x30), "ON", invisible if: CommData.mxRobotOnline
        GroupBox (5,411 344x130), "Request Generator"
            Label (12,18 150x30), "ixAGVatStation"
            Line (10,66) (331,66)
            Lamp1 (177,6 57x53), variable: GVL.ixAGVatStation, style: Lamp-Lamp1-Green
            PushSwitch (257,6 60x58), variable: CommData.mxRequestAGV, behaviour: TOGGLE, style: Switch-PushSwitch-Blue
            Lamp1 (177,73 57x53), variable: CommData.mxNewBookingrequest, style: Lamp-Lamp1-Blue
            PushSwitch (259,70 60x58), variable: CommData.mxNewBookingrequest, behaviour: TOGGLE, style: Switch-PushSwitch-Blue
        GroupBox (173,566 176x126), "Sensor Reading completed", invisible if: NOT CommData.mxWaitingforSensorinput
            PushSwitch (54,26 70x70), variable: CommData.mxScannernoobject, behaviour: TAP, style: Switch-PushSwitch-Red
        GroupBox (2,566 168x127), "Gripper Control"
            Lamp1 (-1748,-553 70x70), style: Lamp-Lamp1-Yellow
            Lamp1 (44,34 70x70), variable: CommData.mxGripper, style: Lamp-Lamp1-Yellow
            RotarySwitch (44,33 70x70), variable: CommData.mxGripper, invisible if: NOT Visualaisation_Control.mxManualMode, behaviour: TOGGLE, style: Switch-RotarySwitch-Blue
        GroupBox (231,27 119x93), "Emergency Stop"
            PushSwitch (23,19 70x70), variable: GVL.ixEmergencyStop, behaviour: TOGGLE, style: Switch-PushSwitch-Red
    Label (900,503 156x30), "Booking from IO Station :"
    Label (650,699 250x30), "Gabriel Sebastian | gabriel.sebastian@hv.se"
END_VISUALIZATION

// ---- VISUs/Visualization.TcVIS
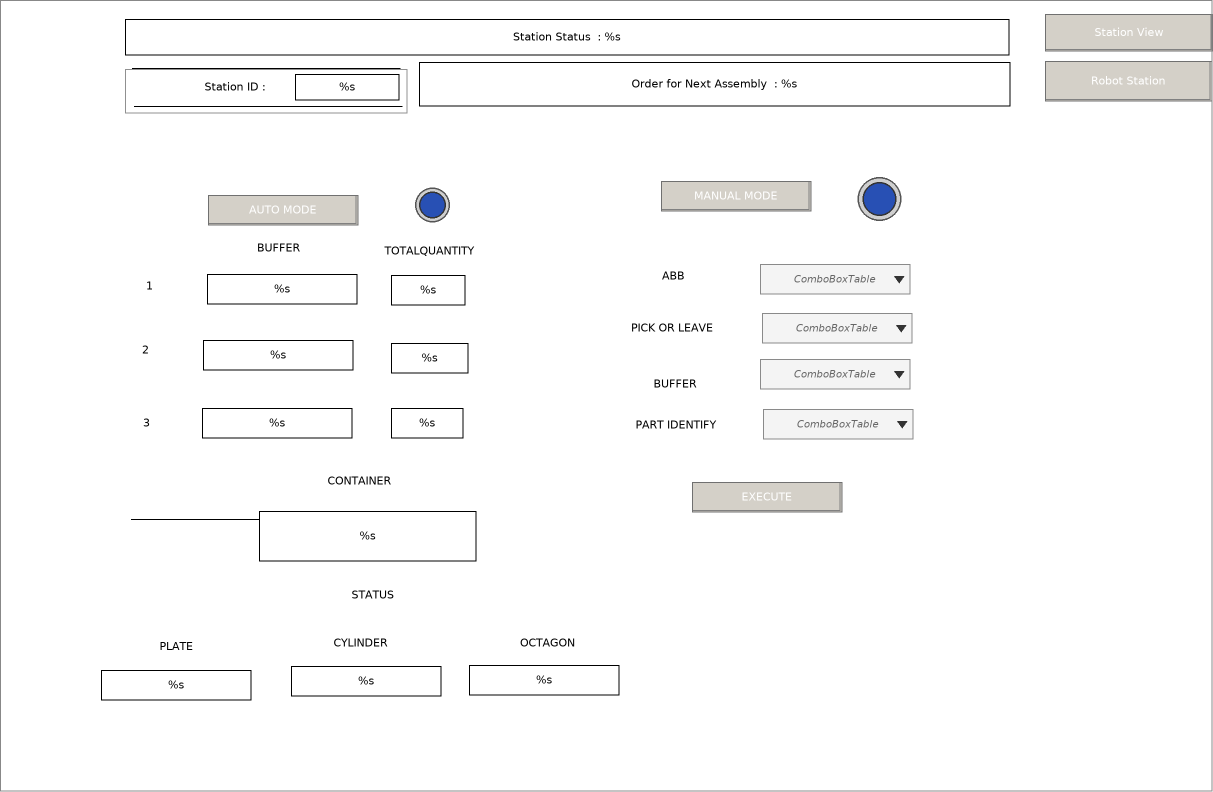
VISUALIZATION Visualization  // 1213x792
    Rectangle (125,19 884x36), "Station Status : %s", text variable: Visualaisation_Control.mxStationStatus
    GroupBox (125,61 282x52)
        Line (6,458) (274,458)
        Line (7,7) (275,7)
        Label (35,11 150x30), "Station ID :"
        Rectangle (170,13 104x26), "%s", text variable: GVL.mwStationID
        Line (9,45) (277,45)
    Button (1045,61 167x40), "Robot Station"
        OnMouseClick: change screen: RobotStation
    Rectangle (419,62 591x44), "Order for Next Assembly : %s", text variable: GVL.qsOrderFornextAssembly
    Button (1045,14 168x37), "Station View"
        OnMouseClick: change screen: Station
    Lamp1 (408,185 49x40), variable: ModeControl.AutoMode, style: Lamp-Lamp1-Blue
    Lamp1 (854,173 51x52), variable: ModeControl.ManualMode, style: Lamp-Lamp1-Blue
    Label (232,233 93x30), "BUFFER"
    Textfield (207,274 150x30), "%s", text variable: GVL.BufferProducts.Storage1.Component
    Label (367,236 125x30), "TOTALQUANTITY"
    Textfield (203,340 150x30), "%s", text variable: GVL.BufferProducts.Storage2.Component
    Textfield (202,408 150x30), "%s", text variable: GVL.BufferProducts.Storage3.Component
    Textfield (391,275 74x30), "%s", text variable: GVL.BufferProducts.Storage1.Quatity
    Textfield (391,343 77x30), "%s", text variable: GVL.BufferProducts.Storage2.Quatity
    Textfield (391,408 72x30), "%s", text variable: GVL.BufferProducts.Storage3.Quatity
    Textfield (259,511 217x50), "%s", text variable: LoadFromAGV.ContainerColor
    Label (133,271 33x30), "1"
    Label (129,335 33x30), "2"
    Label (130,408 33x30), "3"
    Label (296,466 127x30), "CONTAINER"
    Label (118,625 117x43), "PLATE"
    Label (314,628 93x30), "CYLINDER"
    Label (501,628 93x30), "OCTAGON"
    Label (267,575 212x40), "STATUS"
    Label (600,261 150x30), "ABB"
    Label (597,313 150x30), "PICK OR LEAVE"
    Label (600,369 150x30), "BUFFER"
    Label (601,410 150x30), "PART IDENTIFY"
    Label (650,762 150x30)
    Textfield (101,670 150x30), "%s", text variable: AssembleParts.AssembledParts[1]
    Textfield (291,666 150x30), "%s", text variable: AssembleParts.AssembledParts[2]
    Textfield (469,665 150x30), "%s", text variable: AssembleParts.AssembledParts[3]
    Button (692,482 150x30), "EXECUTE"
        tap ManualMode.Execute
    Button (661,181 150x30), "MANUAL MODE"
        tap ModeControl.ManualModeButtonClick
    Button (208,195 150x30), "AUTO MODE"
        tap ModeControl.AutoModeButtonClick
    ComboBoxTable (760,264 150x30), variable: ManualMode.ABBFunction, data array: GVL.sABBFunction
        p3854506369: GVL.sABBFunction[INDEX]
    ComboBoxTable (762,313 150x30), variable: ManualMode.PickLeave, data array: GVL.sPickOrLeave
        p3854506369: GVL.sPickOrLeave[INDEX]
    ComboBoxTable (760,359 150x30), variable: ManualMode.BufferID, data array: GVL.sBufferIDlist
        p3854506369: GVL.sBufferIDlist[INDEX]
    ComboBoxTable (763,409 150x30), variable: ManualMode.Part, data array: GVL.sPart
        p3854506369: GVL.sPart[INDEX]
END_VISUALIZATION
